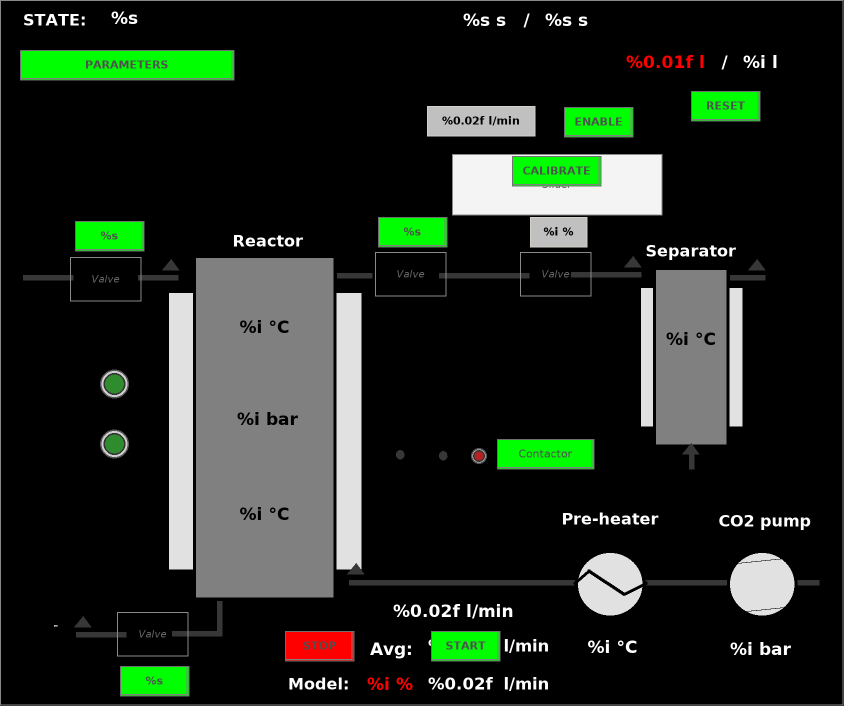
VISUALIZATION ProcessView  // 844x706
    Textfield (390,590 125x42), "%0.02f l/min", text variable: ProcessViewBindings.Co2FlowTextField_TextVariable
    Rectangle (76,632 50x5), colour toggle: ProcessViewBindings.SlurryOutLine1_ToggleColor
    Line (192,441) (126,441)
    Line (192,381) (126,381)
    Rectangle (689,439 5x30)
    Rectangle (419,580 400x5), colour toggle: ProcessViewBindings.ExtractiveOutLines_ToggleColor
    Rectangle (217,601 5x30), colour toggle: ProcessViewBindings.SlurryOutLine1_ToggleColor
    Rectangle (172,631 50x5), colour toggle: ProcessViewBindings.SlurryOutLine1_ToggleColor
    Rectangle (23,275 50x5), colour toggle: ProcessViewBindings.SlurryInArrow_ToggleColor
    Polygon (162,270) (171,259) (179,270) (173,270) (168,270), colour toggle: ProcessViewBindings.SlurryInArrow_ToggleColor
    Rectangle (138,275 40x5), colour toggle: ProcessViewBindings.SlurryInArrow_ToggleColor
    Rectangle (638,285 107x144)
    Rectangle (166,290 198x282), colour toggle: ProcessViewBindings.ReactorBackgroundRectangle_ToggleColor
    RoundedRectangle (193,255 143x345)
    Button (497,439 97x30), "Contactor", colour toggle: ProcessViewBindings.ReactorTemperatureContactorLamp_Variable, invisible if: ProcessViewBindings.ReactorTemperatureContactorButton_Invisible
        toggle ProcessViewBindings.ReactorTemperatureContactorButton_ToggleVariable p2164770859=TRUE
    Lamp1 (465,447 28x18), variable: ProcessViewBindings.ReactorTemperatureContactorLamp_Variable, style: Lamp-Lamp1-Red
    Lamp1 (98,425 33x38), variable: ProcessViewBindings.ReactorLowerLevelLamp, style: Lamp-Lamp1-Green
    Lamp1 (98,365 33x38), variable: ProcessViewBindings.ReactorUpperLevelLamp_Variable, style: Lamp-Lamp1-Green
    Label (193,226 150x30), "Reactor"
    Image (54,625 3x1), image: VisuSymbols.Symbols.TriangleRight
    Button (120,666 69x30), "%s", text variable: ProcessViewBindings.SlurryOutValveButton_TextVariable, colour toggle: ProcessViewBindings.SlurryOutValveButton_ToggleColor, invisible if: ProcessViewBindings.SlurryOutValveButton_Invisible
        toggle ProcessViewBindings.SlurryOutValveButton_ToggleVariable
    Button (75,221 69x30), "%s", text variable: ProcessViewBindings.SlurryInValveControlModeButton_TextVariable, colour toggle: ProcessViewBindings.SlurryInValveControlModeButton_ToggleColor, invisible if: ProcessViewBindings.SlurryInValveControlModeButton_Invisible
        toggle ProcessViewBindings.SlurryInValveControlModeButton_ToggleVariable
    Ellipse (575,550 70x68)
    Polyline (574,584) (589,571) (624,594) (646,583) (644,583)
    Ellipse (727,550 70x68)
    Line (727,564) (785,558)
    Line (727,613) (785,607)
    Label (690,506 150x30), "CO2 pump"
    Label (544,504 132x30), "Pre-heater"
    RoundedRectangle (653,267 76x180)
    Label (616,236 150x30), "Separator"
    Line (396,455) (363,455)
    Ellipse (395,449 10x11)
    Line (438,455) (405,455), invisible if: ProcessViewBindings.ReactorTemperatureContactorClosedLine_Invisible
    Ellipse (438,450 10x11)
    Line (444,440) (411,440), invisible if: ProcessViewBindings.ReactorTemperatureContactorOpenLine_Invisible
    Line (465,455) (447,455)
    Frame (70,257 71x44)
        shows Valve(valve_toggleColor := ProcessViewBindings.SlurryInValveFrame_valve_toggleColor, valve_tapVariable := ProcessViewBindings.SlurryInValveFrame_valve_tapVariable)
    Frame (117,612 71x44)
        shows Valve(valve_toggleColor := ProcessViewBindings.SlurryOutValveFrame_valve_toggleColor, valve_tapVariable := ProcessViewBindings.SlurryOutValveFrame_valve_tapVariable)
    Polygon (74,627) (83,616) (91,627) (85,627) (80,627), colour toggle: ProcessViewBindings.SlurryOutLine1_ToggleColor
    Polygon (347,574) (356,563) (364,574) (358,574) (353,574), colour toggle: ProcessViewBindings.ExtractiveOutLines_ToggleColor
    Rectangle (349,580 75x5), colour toggle: ProcessViewBindings.ExtractiveOutLines_ToggleColor
    Polygon (624,267) (633,256) (641,267) (635,267) (630,267), colour toggle: ProcessViewBindings.ExtractiveOutLines_ToggleColor
    Rectangle (337,273 35x5), colour toggle: ProcessViewBindings.ExtractiveOutLines_ToggleColor
    Polygon (682,454) (691,443) (699,454) (693,454) (688,454)
    Rectangle (730,275 35x5)
    Polygon (748,270) (757,259) (765,270) (759,270) (754,270)
    Rectangle (439,273 90x5), colour toggle: ProcessViewBindings.ExtractiveOutLines_ToggleColor
    Frame (375,252 71x44)
        shows Valve(valve_toggleColor := ProcessViewBindings.ExtractiveOutletOnOff_Valve_ToggleColor, valve_tapVariable := ProcessViewBindings.ExtractiveOutletOnOff_Valve_TapVariable)
    Button (378,217 69x30), "%s", text variable: ProcessViewBindings.ExtractiveOutOnOffValveButton_TextVariable, colour toggle: ProcessViewBindings.ExtractiveOutOnOffValveButton_ToggleColor, invisible if: ProcessViewBindings.ExtractiveOutletOnOff_Valve_Invisible, input disabled if: ProcessViewBindings.ExtractiveOutOnOffValveButton_DisableInputs
        toggle ProcessViewBindings.ExtractiveOutOnOffValveButton_ToggleVariable
    Line (573,242) (524,242)
    Rectangle (571,272 70x5), colour toggle: ProcessViewBindings.ExtractiveOutLines_ToggleColor
    Frame (520,252 71x44)
        shows Valve(valve_toggleColor := ProcessViewBindings.ExtractiveOutletOnOff_Valve_ToggleColor, valve_tapVariable := ProcessViewBindings.ExtractiveOutletOnOff_Valve_TapVariable)
    Slider (452,154 210x61), variable: ProcessViewBindings.ExtractiveOutletValveSlider_Variable, invisible if: TRUE, input disabled if: ProcessViewBindings.ExtractiveOutletValveSlider_DisableInputs, scale 0..10
    Button (20,50 214x30), "PARAMETERS", text variable: ProcessViewBindings.SlurryInValveControlModeButton_TextVariable
        toggle ProcessViewBindings.autoExtractionParameterMenuButton_ToggleVariable
    Textfield (530,217 57x30), "%i %", text variable: ProcessViewBindings.ControlValveOpeningPercentageTextBox_TextVariable, input disabled if: ProcessViewBindings.ControlValveopeningPercentageTextBox_DisableInputs
        OnMouseDown: write ProcessViewBindings.ControlValveOpeningPercentageTextBox_NumPadVariable via VisuDialogs.Numpad, min 0, max 100
    Textfield (209,398 117x42), "%i bar", text variable: ProcessViewBindings.ReactorPressureTextField_TextVariable
    Textfield (206,493 117x42), "%i °C", text variable: ProcessViewBindings.ReactorLowerTemperatureTextField_TextVariable
    Textfield (206,306 117x42), "%i °C", text variable: ProcessViewBindings.ReactorUpperTemperatureTextField_TextVariable
    Textfield (554,626 117x42), "%i °C", text variable: ProcessViewBindings.PreHeaterTemperatureTextField_TextVariable
    Textfield (702,628 117x42), "%i bar", text variable: ProcessViewBindings.Co2PressureTextField_TextVariable
    Textfield (660,318 62x42), "%i °C", text variable: ProcessViewBindings.SeperatorTemperatureTextField_TextVariable
    Label (20,5 81x30), "STATE:"
    Textfield (108,1 310x34), "%s", text variable: ProcessViewBindings.StateLabel_TextVariable
    Textfield (414,3 95x34), "%s s", text variable: ProcessViewBindings.ElapsedTimeLabel_TextVariable, invisible if: ProcessViewBindings.TimeLabels_Invisible
    Textfield (511,3 31x34), "/", invisible if: ProcessViewBindings.TimeLabels_Invisible
    Textfield (542,3 98x34), "%s s", text variable: ProcessViewBindings.CurrentTimeLabel_TextVariable, invisible if: ProcessViewBindings.TimeLabels_Invisible
    Textfield (425,625 125x42), "%0.02f l/min", text variable: ProcessViewBindings.MeanFlowLabel_TextVariable, invisible if: ProcessViewBindings.MeanFlowLabel_Invisible
    Textfield (358,628 58x42), "Avg:"
    Textfield (613,45 95x34), "%0.01f l", text variable: ProcessViewBindings.ConsumedCo2Label_TextVariable
    Textfield (740,45 98x34), "%i l", text variable: ProcessViewBindings.ConsumedCo2SetpointLabel_TextVariable
    Textfield (709,45 31x34), "/"
    Button (691,91 69x30), "RESET"
        tap ProcessViewBindings.ResetCo2ConsumptionButton_TapVariable p3779583253=TRUE
    Button (431,631 69x30), "START", invisible if: ProcessViewBindings.StartMovingAvgCalculationButton_Invisible
        tap ProcessViewBindings.StartMovingAvgCalculationButton_TapVariable p3779583253=TRUE
    Button (285,631 69x30), "STOP", invisible if: ProcessViewBindings.StopMovingAvgCalculationButton_Invisible
        tap ProcessViewBindings.StopMovingAvgCalculationButton_TapVariable p3779583253=TRUE
    Textfield (613,45 95x34), "%0.01f l", text variable: ProcessViewBindings.ConsumedCo2Label_TextVariable, invisible if: ProcessViewBindings.ConsumedCo2alarmLabel_Invisible
    Textfield (285,663 69x42), "Model:", text variable: ProcessViewBindings.Co2FlowTextField_TextVariable, invisible if: ProcessViewBindings.MeanFlowLabel_Invisible
    Textfield (425,663 125x42), "%0.02f l/min", text variable: ProcessViewBindings.Co2ModelLabel_TextVariable, invisible if: ProcessViewBindings.MeanFlowLabel_Invisible
    Textfield (359,663 62x42), "%i %", text variable: ProcessViewBindings.Co2DeviationUnderLimLabel_TextVariable, invisible if: ProcessViewBindings.Co2DeviationUnderLimLabel_Invisible
    Textfield (359,663 62x42), "%i %", text variable: ProcessViewBindings.Co2DeviationUnderLimLabel_TextVariable, invisible if: ProcessViewBindings.Co2DeviationOverLimLabel_Invisible
    Button (512,156 89x30), "CALIBRATE", invisible if: ProcessViewBindings.ExtractiveOutletValveSlider_DisableInputs
        tap ProcessViewBindings.ExtractiveOutletValveCalibrateButton_TapVariable
    Button (564,107 69x30), "ENABLE"
        toggle ProcessViewBindings.MpcEnableButton_ToggleVariable
    Textfield (427,106 108x30), "%0.02f l/min", text variable: ProcessViewBindings.FlowSetPointTextBox_TextVariable
        OnMouseDown: write the text variable via VisuDialogs.Numpad, min 0, max 0.35
END_VISUALIZATION

(* stored: Version 1.1.0.1, ProductVersion 3.1.4024.9
   Visu ProcessView: Id {db42b6b2-d290-49df-811a-85d444c7c9db} *)
